// TIA Portal project "KP8 Driver v2.0 Development" (V15)

(* hardware
DEVICE "S7-1200 station_1"  S7-1200 Station
   slot 0: "Rack_0"  S7-1200 Rack  Rack  V1.0
   slot 1: "PLC_1"  CPU 1211C DC/DC/DC  6ES7 211-1AE40-0XB0  V4.2
DEVICE "HMI_1"  TP700 Comfort Portrait
   slot 0: "HMI_1"  TP700 Comfort Portrait  6AV2 124-0GC01-0AX0  15.0.0.0
   slot 1: "HMI_RT_1"  TP700 Comfort Portrait  6AV2 124-0GC01-0AX0  15.0.0.0
   slot 5: "HMI_1.IE_CP_1"  PROFINET Interface  15.0.0.0
      slot 1: "PROFINET Interface_1"  PROFINET Interface
         slot 1: "Port_1"  Port
         slot 2: "Port_2"  Port
   slot 7: "HMI_1.MPI/DP_CP_1"  MPI/DP Interface  15.0.0.0
*)

// ===== PLC "PLC_1"  CPU 1211C DC/DC/DC =====

VAR_GLOBAL   // PLC tag table "Default tag table"
   "Reset KP8" AT %M100.0 : Bool;
   "Upper/Lower Test" AT %M100.1 : Bool;
   "actual time" AT %MD102 : Time;
   "pulse memory" AT %M100.2 : Bool;
   "inter pulse time" AT %MD104 : Time;
   "State Test" AT %M100.3 : Bool;
   "System_Byte" AT %MB1 : Byte;
   "FirstScan" AT %M1.0 : Bool;
   "DiagStatusUpdate" AT %M1.1 : Bool;
   "AlwaysTRUE" AT %M1.2 : Bool;
   "AlwaysFALSE" AT %M1.3 : Bool;
   "Clock_Byte" AT %MB0 : Byte;
   "Clock_10Hz" AT %M0.0 : Bool;
   "Clock_5Hz" AT %M0.1 : Bool;
   "Clock_2.5Hz" AT %M0.2 : Bool;
   "Clock_2Hz" AT %M0.3 : Bool;
   "Clock_1.25Hz" AT %M0.4 : Bool;
   "Clock_1Hz" AT %M0.5 : Bool;
   "Clock_0.625Hz" AT %M0.6 : Bool;
   "Clock_0.5Hz" AT %M0.7 : Bool;
END_VAR

// folder: KP8

TYPE "KP8 Driver: Button States"
   STRUCT
      btn : Array[0..7] of Bool;
   END_STRUCT;
END_TYPE

TYPE "KP8 Driver: Feedback Data"
   STRUCT
      acutal : "KP8 Driver: Button States";
      falling : "KP8 Driver: Button States";
      rising : "KP8 Driver: Button States";
   END_STRUCT;
END_TYPE

TYPE "KP8 Driver: Parameters: 1 Button"
   STRUCT
      activate : Bool;   // true = button on, flase = button off
      "color on 1" : String[10];   // color when button is in pressed state. valid entries: 'red', 'green', 'blue', 'yellow', 'white', 'off'
      "color on 2" : String[10];   // second flash color when button is pressed and flashing is enabled. valid entries: 'red', 'green', 'blue', 'yellow', 'white', 'off'
      "color off" : String[10];   // color when button is in un-pressed state. valid entries: 'red', 'green', 'blue', 'yellow', 'white', 'off'
      flash : Bool;   // false = color 1, true = color 2. set to clock bit to flash at that rate
      group : Int;   // 0 disables. buttons in groups have a mutually exclusive 'on' state.
      mode : Bool;   // true = maintained, fales = momentary
   END_STRUCT;
END_TYPE

TYPE "KP8 Driver: Parameters: 8 Buttons"
   STRUCT
      btn : Array[0..7] of "KP8 Driver: Parameters: 1 Button";
   END_STRUCT;
END_TYPE

// folder: (top level)

DATA_BLOCK "HMI"   // DB1
{ S7_Optimized_Access := 'TRUE' }
VERSION : 0.1
   VAR
      kp8DQ : DWord;
      kp8DI : Word;
   END_VAR
BEGIN
END_DATA_BLOCK

DATA_BLOCK "KP8 Driver_DB"   // DB2
{ S7_Optimized_Access := 'TRUE' }
VERSION : 2.0
// stored: InstanceOfName KP8 Driver
"KP8 Driver"
BEGIN
END_DATA_BLOCK

DATA_BLOCK "KP8 Button Parameters"   // DB3
{ S7_Optimized_Access := 'TRUE' }
VERSION : 0.1
BEGIN
END_DATA_BLOCK

DATA_BLOCK "KP8 States"   // DB4
{ S7_Optimized_Access := 'TRUE' }
VERSION : 0.1
   VAR
      physical : "KP8 Driver: Feedback Data";
      logical : "KP8 Driver: Feedback Data";
   END_VAR
BEGIN
END_DATA_BLOCK

FUNCTION_BLOCK "KP8 Driver"   // FB1, SCL
{ S7_Optimized_Access := 'TRUE' }
VERSION : 2.0
   VAR_INPUT
      kp8DI : Word;
      reset : Bool;   // resets button states
      btnParams : "KP8 Driver: Parameters: 8 Buttons";
   END_VAR
   VAR_OUTPUT
      kp8DQ : DWord;
      physical : "KP8 Driver: Feedback Data";
      logical : "KP8 Driver: Feedback Data";
   END_VAR
   VAR
      colorMask : DWord;
      old : Struct
         btnParam : "KP8 Driver: Parameters: 8 Buttons";
         kp8DI : Word;
         logical : "KP8 Driver: Button States";
         physical : "KP8 Driver: Button States";
      END_STRUCT;
      btnPress : "KP8 Driver: Button States";
      retLogical : "KP8 Driver: Feedback Data";
   END_VAR
   VAR_TEMP
      color : String;
      draw : Bool;
      pBtn : Int;
      retPhysical : "KP8 Driver: Feedback Data";
      rst : Struct
         feedback : "KP8 Driver: Feedback Data";
         state : "KP8 Driver: Button States";
      END_STRUCT;
   END_VAR
   VAR CONSTANT
      off : DWord := dw#16#0000_0000;
   END_VAR
BEGIN
   REGION "ON RESET REQUEST"
       IF #reset THEN
           #colorMask := #off;
           #old.kp8DI := 16#0;
           #old.logical := #rst.state;
           #old.physical := #rst.state;
           #retPhysical := #rst.feedback;
           #retLogical := #rst.feedback;
           RETURN;
       END_IF;
   END_REGION

   REGION "ON CHANGE IN PARAMETER SET"

       IF #btnParams = #old.btnParam THEN
           GOTO NOUPDATE;
       END_IF;

       REGION "RESET MASK"
           #colorMask := #off;
       END_REGION

       REGION "FOR EACH BUTTON"
           FOR #pBtn := 0 TO 7 DO

               REGION "BUTTON COLOR FOR OFF STATE"
                   IF #btnParams.btn[#pBtn].activate THEN
                       IF NOT #retLogical.acutal.btn[#pBtn] THEN
                           #color := #btnParams.btn[#pBtn]."color off";
                       END_IF;
                   END_IF;
               END_REGION

               REGION "BUTTON COLOR FOR ON STATE"
                   IF #btnParams.btn[#pBtn].activate THEN
                       IF #retLogical.acutal.btn[#pBtn] THEN
                           #color := #btnParams.btn[#pBtn]."color on 1";
                       END_IF;
                   END_IF;
               END_REGION

               REGION "DEACTIVATED BUTTON"
                   (*
                   This is here for redundancy.
                   The "RESET MASK" region takes care of clearing old button colors.
                   *)
                   IF NOT #btnParams.btn[#pBtn].activate THEN
                       #color := 'OFF';
                   END_IF;
               END_REGION

               REGION "DRAW COLOR"
                   "KP8 Driver: Color"(btnColor := #colorMask,
                                       btnNum := #pBtn,
                                       lblColor := #color);
               END_REGION

           END_FOR;
       END_REGION

   END_REGION

   NOUPDATE:

   REGION "FEEDBACK"

       REGION "SCATTER KP8 INPUT BYTE"
           SCATTER(IN := #kp8DI.%B1,
                   OUT => #btnPress.btn);
       END_REGION

       REGION "FOR EACH BUTTON"
           FOR #pBtn := 0 TO 7 DO

               REGION "PHYSICAL FEEDBACK"
                   "KP8 Driver: Feedback"(signal := #btnPress.btn[#pBtn],
                                          oldSignal := #old.physical.btn[#pBtn],
                                          btnNumber := #pBtn,
                                          feedback := #retPhysical);
               END_REGION

               REGION "DETERMINE LOGICAL STATE"
                   "KP8 Driver: State"(press := #retPhysical,
                                       btnNumber := #pBtn,
                                       btnParams := #btnParams,
                                       state := #retLogical);
               END_REGION



           END_FOR;
       END_REGION

       REGION "FOR EACH BUTTON: LOGICAL FEEDBACK"
           (*
           this needs a separate loop so that group exclusivity can be evaluated
           properly.
           *)
           FOR #pBtn := 0 TO 7 DO
               "KP8 Driver: Feedback"(signal := #retLogical.acutal.btn[#pBtn],
                                      oldSignal := #old.logical.btn[#pBtn],
                                      btnNumber := #pBtn,
                                      feedback := #retLogical);
           END_FOR;
       END_REGION

   END_REGION

   REGION "ANIMATE BUTTONS"

       REGION "FOR EACH BUTTON"
           FOR #pBtn := 0 TO 7 DO

               REGION "CHANGE COLOR TO ON 1" 
                   IF #retLogical.rising.btn[#pBtn] THEN
                       #color := #btnParams.btn[#pBtn]."color on 1";
                       #draw := TRUE;
                   END_IF;
               END_REGION

               REGION "CHANGE COLOR TO OFF" 
                   IF #retLogical.falling.btn[#pBtn] THEN
                       #color := #btnParams.btn[#pBtn]."color off";
                       #draw := TRUE;
                   END_IF;
               END_REGION

               REGION "FLASHING"
                   IF #retLogical.acutal.btn[#pBtn] THEN

                       REGION "FLASH COLOR 1"
                           IF NOT #btnParams.btn[#pBtn].flash THEN
                               IF #old.btnParam.btn[#pBtn].flash THEN
                                   #color := #btnParams.btn[#pBtn]."color on 1";
                                   #draw := TRUE;
                               END_IF;
                           END_IF;
                       END_REGION

                       REGION "FLASH COLOR 2"
                           IF #btnParams.btn[#pBtn].flash THEN
                               IF NOT #old.btnParam.btn[#pBtn].flash THEN
                                   #color := #btnParams.btn[#pBtn]."color on 2";
                                   #draw := TRUE;
                               END_IF;
                           END_IF;
                       END_REGION

                   END_IF;
               END_REGION

               REGION "DRAW TO BUTTON"
                   IF #draw THEN
                       #draw := FALSE;
                       "KP8 Driver: Color"(btnColor := #colorMask,
                                           btnNum := #pBtn,
                                           lblColor := #color);
                   END_IF;
               END_REGION

           END_FOR;
       END_REGION

   END_REGION

   REGION "CHANGE DETECTION"
       #old.btnParam := #btnParams;
       #old.kp8DI := #kp8DI;
       #old.logical := #retLogical.acutal;
       #old.physical := #btnPress;
   END_REGION

   REGION "OUTPUT"
       #kp8DQ := #colorMask;
       #physical := #retPhysical;
       #logical := #retLogical;
   END_REGION
END_FUNCTION_BLOCK

FUNCTION "KP8 Driver: Group" : Void   // FC1, SCL
{ S7_Optimized_Access := 'TRUE' }
VERSION : 0.1
   VAR_INPUT
      btnNumber : Int;
      btnsParams : "KP8 Driver: Parameters: 8 Buttons";
   END_VAR
   VAR_IN_OUT
      logical : "KP8 Driver: Feedback Data";
   END_VAR
   VAR_TEMP
      pBtn : Int;
      retLogical : "KP8 Driver: Feedback Data";
      testGroup : Int;
      thisGroup : Int;
   END_VAR
BEGIN
   REGION "EXIT IF GROUP EQUALS 0"
       #thisGroup := #btnsParams.btn[#btnNumber].group;
       IF #thisGroup = 0 THEN
           RETURN;
       END_IF;
   END_REGION

   REGION "COPY TO LOCAL"
       #retLogical := #logical;
   END_REGION

   REGION "FOR EACH BUTTONS' PARAMETERS"
       FOR #pBtn := 0 TO 7 DO

           REGION "SKIP THE CURRENT BUTTON"
               IF #pBtn = #btnNumber THEN
                   GOTO NEXT;
               END_IF;
           END_REGION

           REGION "GROUP EXCLUSION"
               #testGroup := #btnsParams.btn[#pBtn].group;
               IF #testGroup = #thisGroup THEN
                   #retLogical.acutal.btn[#pBtn] := FALSE;
               END_IF;
           END_REGION

       NEXT:
           ;

       END_FOR;
   END_REGION

   REGION "OUTPUT"
       #logical := #retLogical;
   END_REGION
END_FUNCTION

FUNCTION "KP8 Driver: Toggle" : Void   // FC2, SCL
{ S7_Optimized_Access := 'TRUE' }
VERSION : 0.1
   VAR_INPUT
      signal : Bool;   // edge signal
   END_VAR
   VAR_IN_OUT
      state : Bool;   // logical button state
   END_VAR
BEGIN
   IF #signal THEN
       #state := NOT #state;
   END_IF;
END_FUNCTION

FUNCTION "KP8 Driver: State" : Void   // FC3, SCL
{ S7_Optimized_Access := 'TRUE' }
VERSION : 0.1
   VAR_INPUT
      press : "KP8 Driver: Feedback Data";
      btnNumber : Int;
      btnParams : "KP8 Driver: Parameters: 8 Buttons";
   END_VAR
   VAR_IN_OUT
      state : "KP8 Driver: Feedback Data";
   END_VAR
   VAR_TEMP
      pBtn : Int;
      retState : "KP8 Driver: Feedback Data";
   END_VAR
BEGIN
   REGION "RETURN ON INACTIVE BUTTON"
       IF NOT #btnParams.btn[#btnNumber].activate THEN
           RETURN;
       END_IF;
   END_REGION

   REGION "COPY TO LOCAL"
       #retState := #state;
   END_REGION

   REGION "MODE IS MOMENTARY"
       IF NOT #btnParams.btn[#btnNumber].mode THEN
           #retState.acutal.btn[#btnNumber] := #press.acutal.btn[#btnNumber];
       END_IF;
   END_REGION

   REGION "MAINTINED"
       IF #btnParams.btn[#btnNumber].mode THEN
           "KP8 Driver: Toggle"(signal := #press.rising.btn[#btnNumber],
                                state := #retState.acutal.btn[#btnNumber]);
       END_IF;
   END_REGION

   REGION "GROUP EXCLUSIVITY"
       IF #press.rising.btn[#btnNumber] THEN
           "KP8 Driver: Group"(btnNumber := #btnNumber,
                               btnsParams := #btnParams,
                               logical := #retState);
       END_IF;
   END_REGION

   REGION "OUTPUT"
       #state := #retState;
   END_REGION
END_FUNCTION

FUNCTION "KP8 Driver: Feedback" : Void   // FC4, SCL
{ S7_Optimized_Access := 'TRUE' }
VERSION : 0.1
   VAR_INPUT
      signal : Bool;
      oldSignal : Bool;
      btnNumber : Int;
   END_VAR
   VAR_IN_OUT
      feedback : "KP8 Driver: Feedback Data";
   END_VAR
   VAR_TEMP
      ret : "KP8 Driver: Feedback Data";
   END_VAR
BEGIN
   REGION "COPY TO LOCAL"
       #ret := #feedback;
       #ret.acutal.btn[#btnNumber] := #signal;
   END_REGION

   REGION "DEFAULT"
       #ret.rising.btn[#btnNumber] := FALSE;
       #ret.falling.btn[#btnNumber] := FALSE;
   END_REGION

   REGION "ON NEW INPUT"
       IF #signal <> #oldSignal THEN

           REGION "RISING EDGE"
               IF #signal AND NOT #oldSignal THEN
                   #ret.rising.btn[#btnNumber] := TRUE;
               END_IF;
           END_REGION

           REGION "FALLING EDGE"
               IF NOT #signal AND #oldSignal THEN
                   #ret.falling.btn[#btnNumber] := TRUE;
               END_IF;
           END_REGION

       END_IF;
   END_REGION


   REGION "OUTPUT"
       #feedback := #ret;
   END_REGION
END_FUNCTION

FUNCTION "Upper" : Void   // FC5, SCL
{ S7_Optimized_Access := 'TRUE' }
VERSION : 0.1
   VAR_IN_OUT
      "string" : Variant;
   END_VAR
   VAR_TEMP
      "type" : Bool;
      stringBox : String;
      status : Int;
      wStringBox : WString;
      charArr : Array[0..255] of Char;
      cntChar : UInt;
      pChar : Int;
   END_VAR
   VAR CONSTANT
      asciiLow : Char := 'a';
      asciiHigh : Char := 'z';
      asciiCaseOffset : Int := 32;
   END_VAR
BEGIN
   IF TypeOf(#string) = String THEN
       #status := MOVE_BLK_VARIANT(SRC := #string,
                                   COUNT := 1,
                                   SRC_INDEX := 0,
                                   DEST_INDEX := 0,
                                   DEST => #stringBox);
   ELSIF TypeOf(#string) = WString THEN
       #status := MOVE_BLK_VARIANT(SRC := #string,
                                   COUNT := 1,
                                   SRC_INDEX := 0,
                                   DEST_INDEX := 0,
                                   DEST => #wStringBox);
       #stringBox := WSTRING_TO_STRING(#wStringBox);
   ELSE
       RETURN;
   END_IF;

   Strg_TO_Chars(Strg := #stringBox,
                 pChars := 0,
                 Cnt => #cntChar,
                 Chars := #charArr);

   FOR #pChar := 0 TO UINT_TO_INT(#cntChar) - 1 DO
       IF #asciiLow <= #charArr[#pChar] AND #charArr[#pChar] <= #asciiHigh THEN
           #charArr[#pChar] := INT_TO_CHAR(CHAR_TO_INT(#charArr[#pChar]) - #asciiCaseOffset);
       END_IF;
   END_FOR;

   Chars_TO_Strg(Chars := #charArr,
                 pChars := 0,
                 Cnt := #cntChar,
                 Strg => #stringBox);

   IF TypeOf(#string) = String THEN
       #status := MOVE_BLK_VARIANT(SRC := #stringBox,
                                   COUNT := 1,
                                   SRC_INDEX := 0,
                                   DEST_INDEX := 0,
                                   DEST => #string);
   ELSIF TypeOf(#string) = WString THEN
       #wStringBox := STRING_TO_WSTRING(#stringBox);
       #status := MOVE_BLK_VARIANT(SRC := #wStringBox,
                                   COUNT := 1,
                                   SRC_INDEX := 0,
                                   DEST_INDEX := 0,
                                   DEST => #string);
   END_IF;
END_FUNCTION

FUNCTION "KP8 Driver: Color" : Void   // FC38, SCL
{ S7_Optimized_Access := 'TRUE' }
VERSION : 0.1
   VAR_INPUT
      btnNum : Int;
      lblColor : String;
   END_VAR
   VAR_IN_OUT
      btnColor : DWord;
   END_VAR
   VAR_TEMP
      btnMask : DWord;
      uColor : String;
      ret : DWord;
   END_VAR
   VAR CONSTANT
      btnMskRed : DWord := dw#16#0100_0000;
      btnMskGreen : DWord := dw#16#0001_0000;
      btnMskBlue : DWord := dw#16#000_0100;
      btnMskYellow : DWord := dw#16#0101_0000;
      btnMskWhite : DWord := dw#16#0101_0100;
      btnMskOff : DWord := dw#16#FEFE_FEFF;
   END_VAR
BEGIN
   #ret := #btnColor;

   #ret := #ret AND ROL(IN := #btnMskOff,
                        N := INT_TO_UDINT(#btnNum));

   #uColor := #lblColor;
   "Upper"(#uColor);

   IF (#uColor = 'RED') THEN
       #btnMask := #btnMskRed;
   ELSIF (#uColor = 'GREEN') THEN
       #btnMask := #btnMskGreen;
   ELSIF (#uColor = 'BLUE') THEN
       #btnMask := #btnMskBlue;
   ELSIF (#uColor = 'YELLOW') THEN
       #btnMask := #btnMskYellow;
   ELSIF (#uColor = 'WHITE') THEN
       #btnMask := #btnMskWhite;
   ELSIF (#uColor = 'OFF') THEN
       ;
   END_IF;

   #ret := #ret OR SHL(IN := #btnMask,
                       N := INT_TO_UDINT(#btnNum));

   #btnColor := #ret;
END_FUNCTION

ORGANIZATION_BLOCK "Main"   // OB1, LAD, ProgramCycle
TITLE = "Main Program Sweep (Cycle)"
{ S7_Optimized_Access := 'TRUE' }
VERSION : 0.1
   VAR_INPUT
      Initial_Call : Bool;   // Initial call of this OB
      Remanence : Bool;   // =True, if remanent data are available
   END_VAR
BEGIN

REGION Network 1
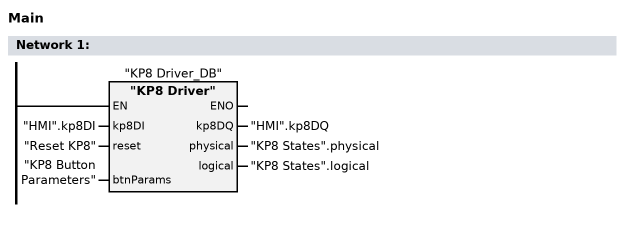
   RUNG wire#powerrail
      "KP8 Driver_DB"(kp8DI := "HMI".kp8DI, reset := "Reset KP8", btnParams := "KP8 Button Parameters", kp8DQ => "HMI".kp8DQ, physical => "KP8 States".physical, logical => "KP8 States".logical)
   END_RUNG
   // the same network as SCL:
   "KP8 Driver_DB"(kp8DI := "HMI".kp8DI,   // "KP8 Driver"
                   reset := "Reset KP8",
                   btnParams := "KP8 Button Parameters",
                   kp8DQ => "HMI".kp8DQ,
                   physical => "KP8 States".physical,
                   logical => "KP8 States".logical);
END_REGION
END_ORGANIZATION_BLOCK

(* ===== HMI "HMI_RT_1" =====
system functions are stored by id; their names below are inferred from use
connection "HMI_Connection_1": ETHERNET, S7_1200_OMS

HMI tags "Default tag table"
   "HMI_kp8DQ" : DWord = PLC HMI.kp8DQ AT %DB1.DBW0, 100 ms
      on ChangeValue: "parseKP8DQ"("HMI_kp8DQ")
   "HMI_kp8DI" : Word = PLC HMI.kp8DI AT %DB1.DBD0, 100 ms
   "key0Color" : UDInt AT %DB1.DBW0
   "key1Color" : UDInt AT %DB1.DBD0
   "key2Color" : UDInt, internal
   "key3Color" : UDInt, internal
   "key4Color" : UDInt, internal
   "key5Color" : UDInt, internal
   "key6Color" : UDInt, internal
   "key7Color" : UDInt, internal

screen "KP8" 480x800
   Button "btnKP7Btn7" at 121,147 size 103x103; TextOff '7'
      Appearance <- "key7Color"
      on Press: function_b14e0dd5("HMI_kp8DI", 15)
   Button "btnKP7Btn3" at 255,147 size 103x103; TextOff '3'
      Appearance <- "key3Color"
      on Press: function_b14e0dd5("HMI_kp8DI", 11)
   Button "btnKP7Btn6" at 121,281 size 103x103; TextOff '6'
      Appearance <- "key6Color"
      on Press: function_b14e0dd5("HMI_kp8DI", 14)
   Button "btnKP7Btn2" at 255,281 size 103x103; TextOff '2'
      Appearance <- "key2Color"
      on Press: function_b14e0dd5("HMI_kp8DI", 10)
   Button "btnKP7Btn5" at 121,415 size 103x103; TextOff '5'
      Appearance <- "key5Color"
      on Press: function_b14e0dd5("HMI_kp8DI", 13)
   Button "btnKP7Btn1" at 255,415 size 103x103; TextOff '1'
      Appearance <- "key1Color"
      on Press: function_b14e0dd5("HMI_kp8DI", 9)
   Button "btnKP7Btn4" at 121,549 size 103x103; TextOff '4'
      Appearance <- "key4Color"
      on Press: function_b14e0dd5("HMI_kp8DI", 12)
   Button "btnKP7Btn0" at 255,549 size 103x103; TextOff '0'
      Appearance <- "key0Color"
      on Press: function_b14e0dd5("HMI_kp8DI", 8)
   IOField "I/O field_1" at 260,554 size 93x20; FormatPattern FFFFFF
      ProcessValue <- "key0Color"
      Appearance <- "key0Color"
   IOField "I/O field_2" at 260,420 size 93x20; FormatPattern FFFFFF
      ProcessValue <- "key1Color"
      Appearance <- "key1Color"
   IOField "I/O field_3" at 260,286 size 93x20; FormatPattern FFFFFF
      ProcessValue <- "key2Color"
      Appearance <- "key2Color"
   IOField "I/O field_4" at 260,152 size 93x20; FormatPattern FFFFFF
      ProcessValue <- "key3Color"
      Appearance <- "key3Color"
   IOField "I/O field_5" at 126,554 size 93x20; FormatPattern FFFFFF
      ProcessValue <- "key4Color"
      Appearance <- "key4Color"
   IOField "I/O field_6" at 126,420 size 93x20; FormatPattern FFFFFF
      ProcessValue <- "key5Color"
      Appearance <- "key5Color"
   IOField "I/O field_7" at 126,286 size 93x20; FormatPattern FFFFFF
      ProcessValue <- "key6Color"
      Appearance <- "key6Color"
   IOField "I/O field_8" at 126,152 size 93x20; FormatPattern FFFFFF
      ProcessValue <- "key7Color"
      Appearance <- "key7Color"
   IOField "I/O field_9" at 49,95 size 382x50; FormatPattern FFFFFFFF
      ProcessValue <- "HMI_kp8DQ"

VB script "shiftLeft"
   	Dim ret 
   	ret = Int(kp8DQ / 2^8)
   	ret = Int(ret / 2^pBtn)
   	ret = ret And 65793
   	shiftLeft = ret

VB script "parseKP8DQ"
   	Dim pBtn	
   	For pBtn = 0 To 7
   		SmartTags("key"&pBtn&"Color") = shiftLeft(kp8DQ,pBtn)
   	Next
*)